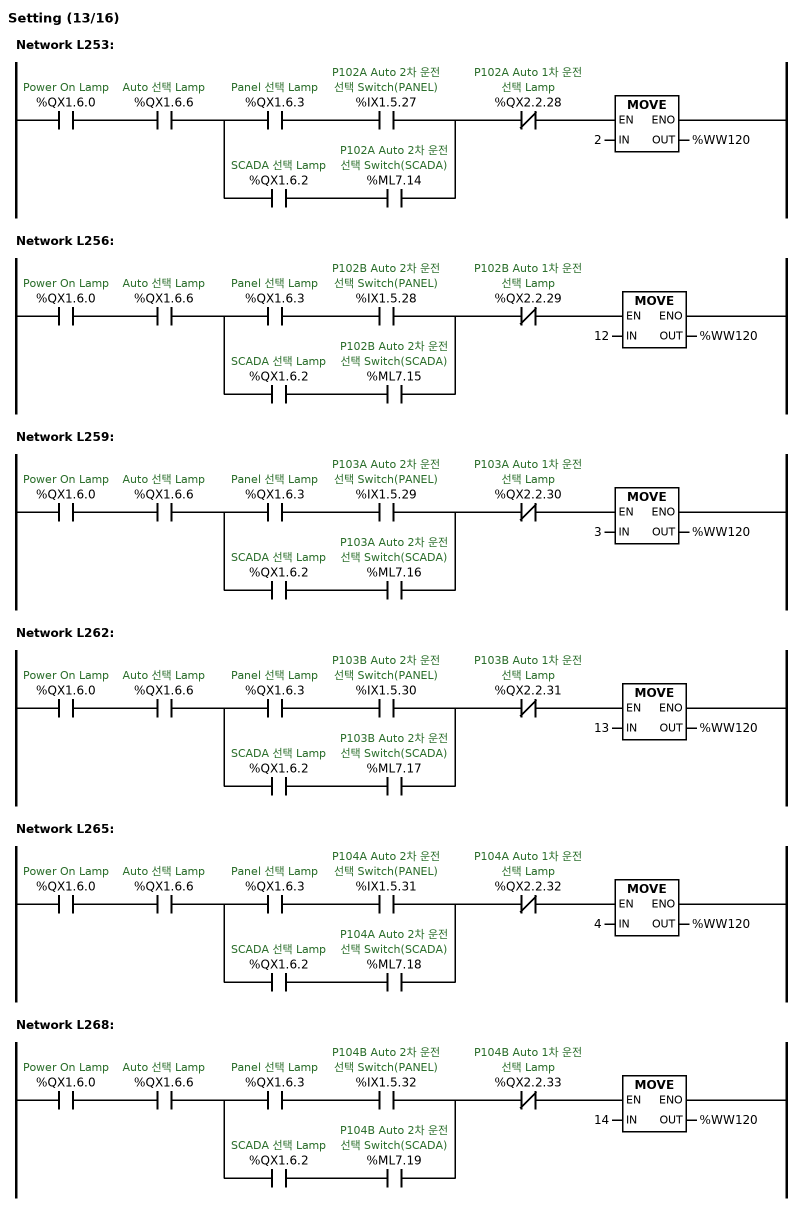
(* [picture p144: Setting rungs L253-L268] *)
(* Rung L253 *)
IF %QX1.6.0 AND %QX1.6.6 AND ((%QX1.6.3 AND %IX1.5.27) OR (%QX1.6.2 AND %ML7.14)) AND NOT %QX2.2.28 THEN
    %WW120 := 2;
END_IF;
(* Rung L256 *)
IF %QX1.6.0 AND %QX1.6.6 AND ((%QX1.6.3 AND %IX1.5.28) OR (%QX1.6.2 AND %ML7.15)) AND NOT %QX2.2.29 THEN
    %WW120 := 12;
END_IF;
(* Rung L259 *)
IF %QX1.6.0 AND %QX1.6.6 AND ((%QX1.6.3 AND %IX1.5.29) OR (%QX1.6.2 AND %ML7.16)) AND NOT %QX2.2.30 THEN
    %WW120 := 3;
END_IF;
(* Rung L262 *)
IF %QX1.6.0 AND %QX1.6.6 AND ((%QX1.6.3 AND %IX1.5.30) OR (%QX1.6.2 AND %ML7.17)) AND NOT %QX2.2.31 THEN
    %WW120 := 13;
END_IF;
(* Rung L265 *)
IF %QX1.6.0 AND %QX1.6.6 AND ((%QX1.6.3 AND %IX1.5.31) OR (%QX1.6.2 AND %ML7.18)) AND NOT %QX2.2.32 THEN
    %WW120 := 4;
END_IF;
(* Rung L268 *)
IF %QX1.6.0 AND %QX1.6.6 AND ((%QX1.6.3 AND %IX1.5.32) OR (%QX1.6.2 AND %ML7.19)) AND NOT %QX2.2.33 THEN
    %WW120 := 14;
END_IF;

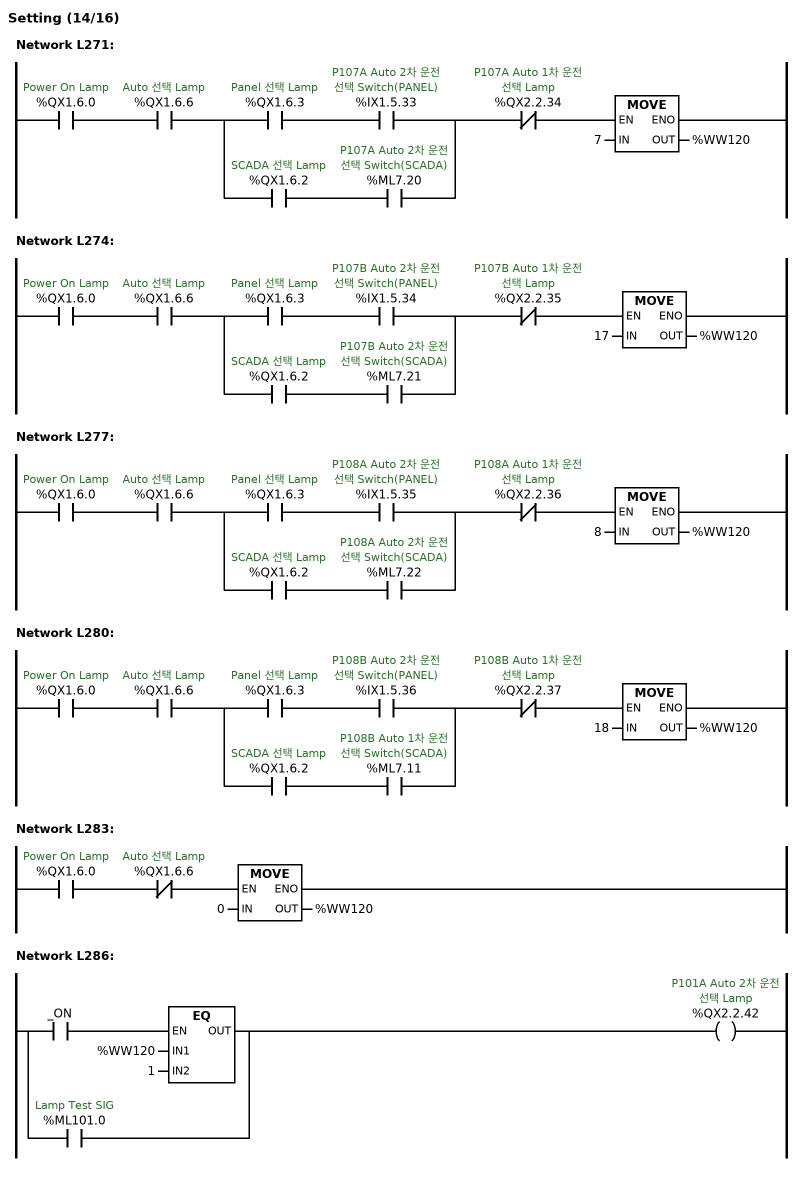
(* Rung L271 *)
IF %QX1.6.0 AND %QX1.6.6 AND ((%QX1.6.3 AND %IX1.5.33) OR (%QX1.6.2 AND %ML7.20)) AND NOT %QX2.2.34 THEN
    %WW120 := 7;
END_IF;
(* Rung L274 *)
IF %QX1.6.0 AND %QX1.6.6 AND ((%QX1.6.3 AND %IX1.5.34) OR (%QX1.6.2 AND %ML7.21)) AND NOT %QX2.2.35 THEN
    %WW120 := 17;
END_IF;
(* Rung L277 *)
IF %QX1.6.0 AND %QX1.6.6 AND ((%QX1.6.3 AND %IX1.5.35) OR (%QX1.6.2 AND %ML7.22)) AND NOT %QX2.2.36 THEN
    %WW120 := 8;
END_IF;
(* Rung L280 *)
IF %QX1.6.0 AND %QX1.6.6 AND ((%QX1.6.3 AND %IX1.5.36) OR (%QX1.6.2 AND %ML7.11)) AND NOT %QX2.2.37 THEN
    %WW120 := 18;
END_IF;
(* Rung L283 *)
IF %QX1.6.0 AND NOT %QX1.6.6 THEN %WW120 := 0; END_IF;
(* Rung L286 *)
IF _ON THEN _t23 := %WW120 = 1; END_IF;
%QX2.2.42 := _t23 OR %ML101.0;

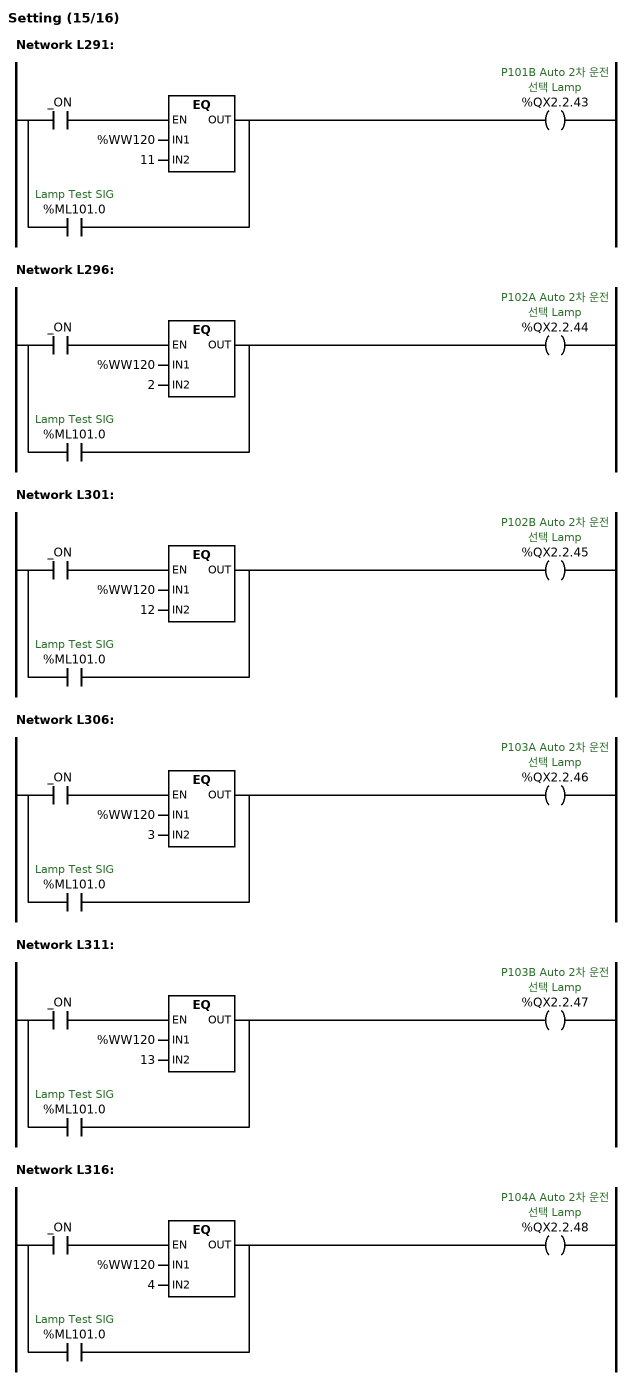
(* Rung L291 *)
IF _ON THEN _t24 := %WW120 = 11; END_IF;
%QX2.2.43 := _t24 OR %ML101.0;
(* Rung L296 *)
IF _ON THEN _t25 := %WW120 = 2; END_IF;
%QX2.2.44 := _t25 OR %ML101.0;
(* Rung L301 *)
IF _ON THEN _t26 := %WW120 = 12; END_IF;
%QX2.2.45 := _t26 OR %ML101.0;
(* Rung L306 *)
IF _ON THEN _t27 := %WW120 = 3; END_IF;
%QX2.2.46 := _t27 OR %ML101.0;
(* Rung L311 *)
IF _ON THEN _t28 := %WW120 = 13; END_IF;
%QX2.2.47 := _t28 OR %ML101.0;
(* Rung L316 *)
IF _ON THEN _t29 := %WW120 = 4; END_IF;
%QX2.2.48 := _t29 OR %ML101.0;

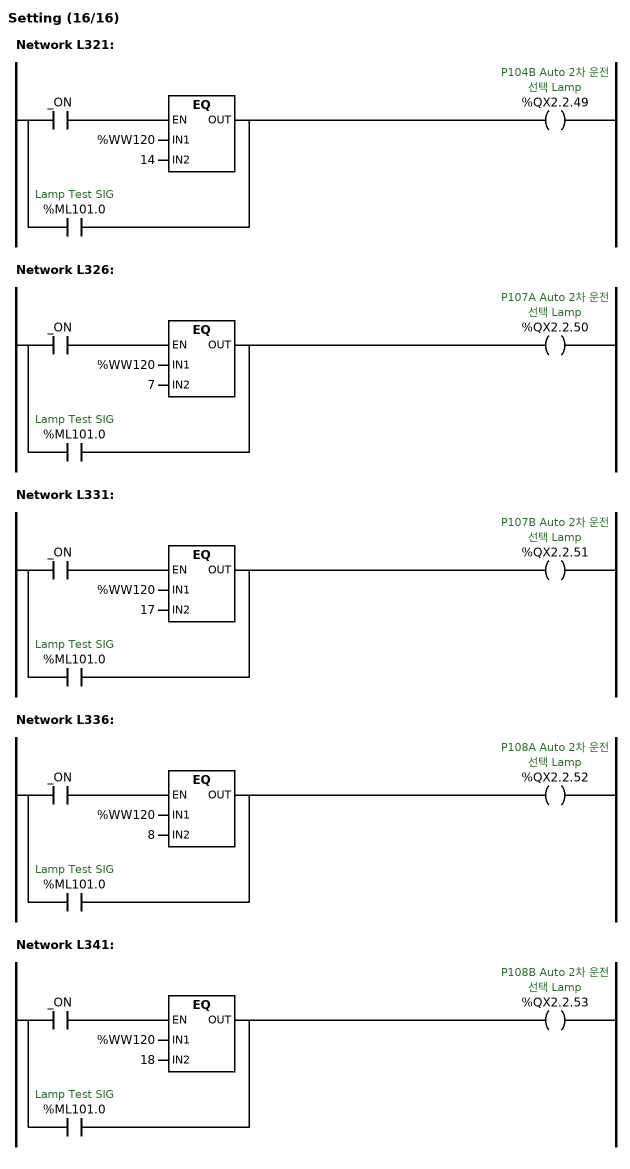
(* Rung L321 *)
IF _ON THEN _t30 := %WW120 = 14; END_IF;
%QX2.2.49 := _t30 OR %ML101.0;
(* Rung L326 *)
IF _ON THEN _t31 := %WW120 = 7; END_IF;
%QX2.2.50 := _t31 OR %ML101.0;
(* Rung L331 *)
IF _ON THEN _t32 := %WW120 = 17; END_IF;
%QX2.2.51 := _t32 OR %ML101.0;
(* Rung L336 *)
IF _ON THEN _t33 := %WW120 = 8; END_IF;
%QX2.2.52 := _t33 OR %ML101.0;
(* Rung L341 *)
IF _ON THEN _t34 := %WW120 = 18; END_IF;
%QX2.2.53 := _t34 OR %ML101.0;
END_PROGRAM

PROGRAM Alarm (* task: 스캔 프로그램 *)
VAR
    _e1 : R_TRIG;
    _e2 : R_TRIG;
    _e3 : R_TRIG;
    _e4 : R_TRIG;
    _e5 : R_TRIG;
    _e6 : R_TRIG;
    _e7 : R_TRIG;
    _e8 : R_TRIG;
END_VAR

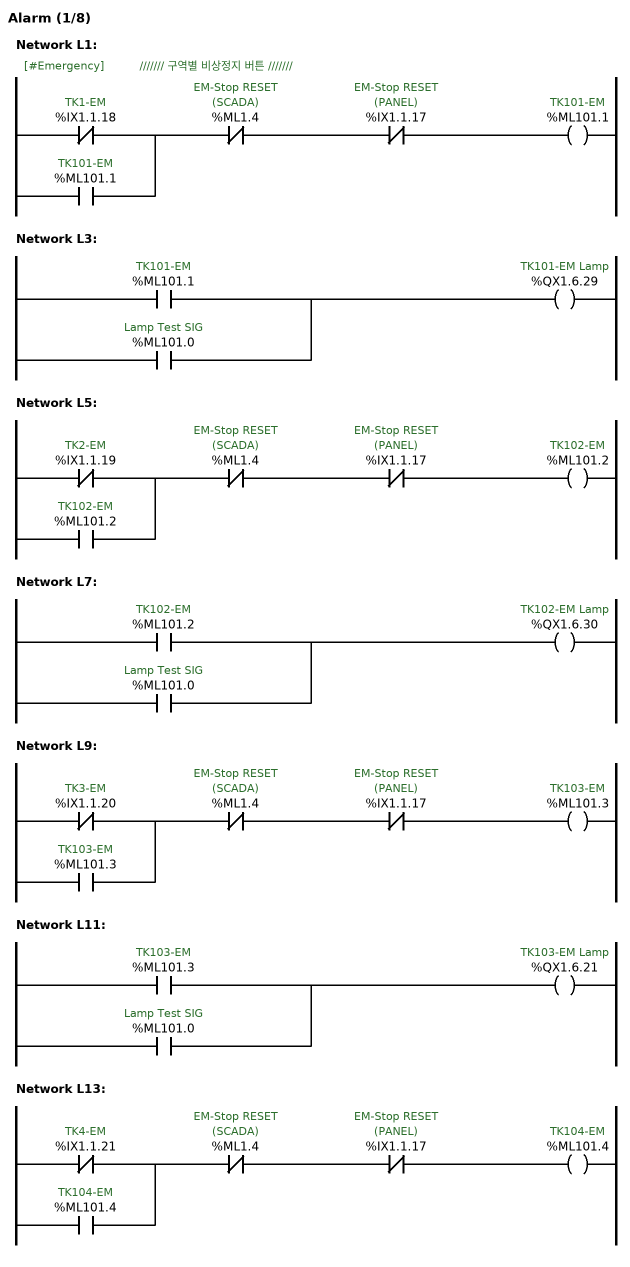
(* [#Emergency]          /////// 구역별 비상정지 버튼 /////// *)
(* Rung L1 *)
%ML101.1 := (NOT %IX1.1.18 OR %ML101.1) AND NOT %ML1.4 AND NOT %IX1.1.17;
(* Rung L3 *)
%QX1.6.29 := %ML101.1 OR %ML101.0;
(* Rung L5 *)
%ML101.2 := (NOT %IX1.1.19 OR %ML101.2) AND NOT %ML1.4 AND NOT %IX1.1.17;
(* Rung L7 *)
%QX1.6.30 := %ML101.2 OR %ML101.0;
(* Rung L9 *)
%ML101.3 := (NOT %IX1.1.20 OR %ML101.3) AND NOT %ML1.4 AND NOT %IX1.1.17;
(* Rung L11 *)
%QX1.6.21 := %ML101.3 OR %ML101.0;
(* Rung L13 *)
%ML101.4 := (NOT %IX1.1.21 OR %ML101.4) AND NOT %ML1.4 AND NOT %IX1.1.17;

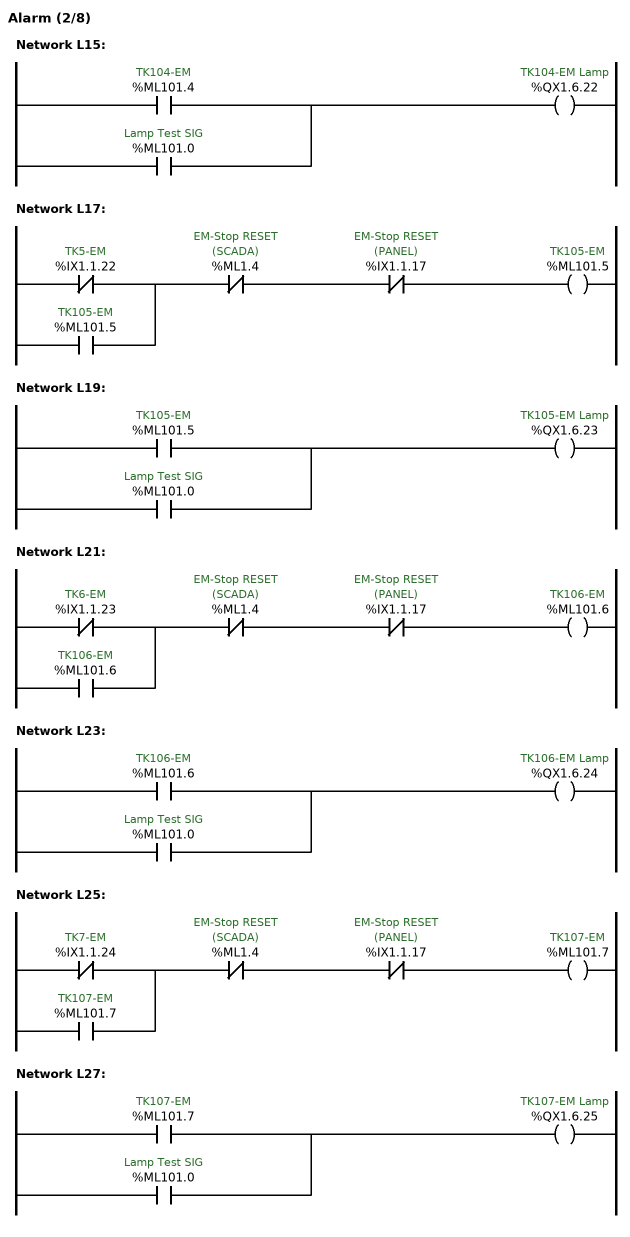
(* Rung L15 *)
%QX1.6.22 := %ML101.4 OR %ML101.0;
(* Rung L17 *)
%ML101.5 := (NOT %IX1.1.22 OR %ML101.5) AND NOT %ML1.4 AND NOT %IX1.1.17;
(* Rung L19 *)
%QX1.6.23 := %ML101.5 OR %ML101.0;
(* Rung L21 *)
%ML101.6 := (NOT %IX1.1.23 OR %ML101.6) AND NOT %ML1.4 AND NOT %IX1.1.17;
(* Rung L23 *)
%QX1.6.24 := %ML101.6 OR %ML101.0;
(* Rung L25 *)
%ML101.7 := (NOT %IX1.1.24 OR %ML101.7) AND NOT %ML1.4 AND NOT %IX1.1.17;
(* Rung L27 *)
%QX1.6.25 := %ML101.7 OR %ML101.0;

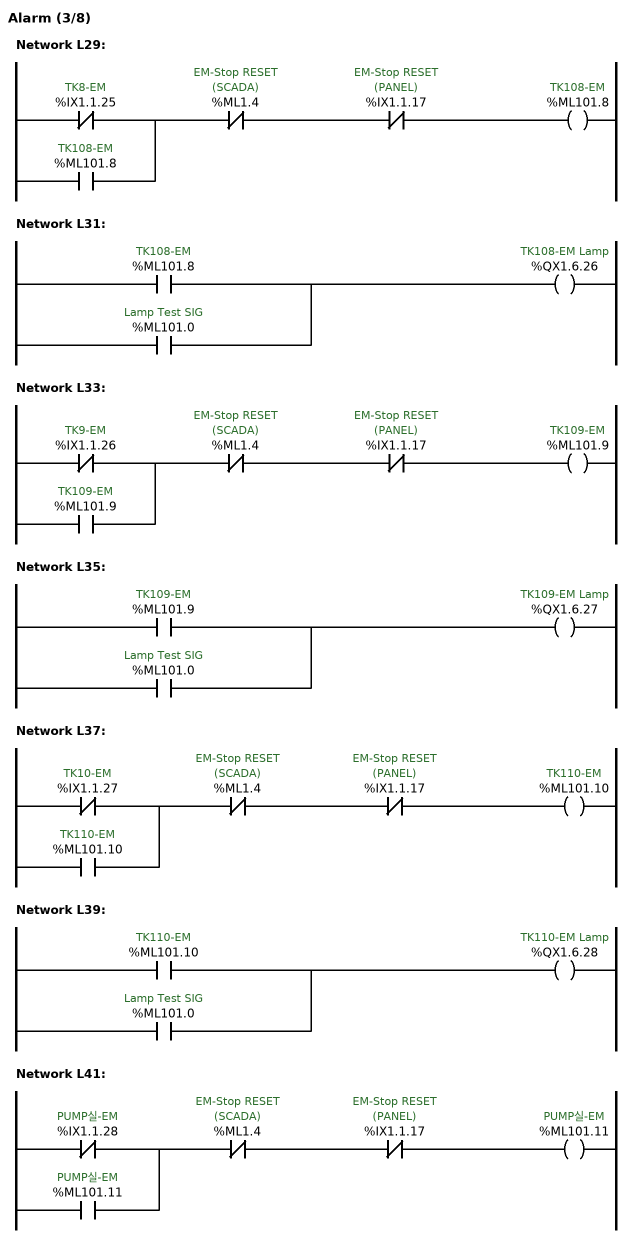
(* Rung L29 *)
%ML101.8 := (NOT %IX1.1.25 OR %ML101.8) AND NOT %ML1.4 AND NOT %IX1.1.17;
(* Rung L31 *)
%QX1.6.26 := %ML101.8 OR %ML101.0;
(* Rung L33 *)
%ML101.9 := (NOT %IX1.1.26 OR %ML101.9) AND NOT %ML1.4 AND NOT %IX1.1.17;
(* Rung L35 *)
%QX1.6.27 := %ML101.9 OR %ML101.0;
(* Rung L37 *)
%ML101.10 := (NOT %IX1.1.27 OR %ML101.10) AND NOT %ML1.4 AND NOT %IX1.1.17;
(* Rung L39 *)
%QX1.6.28 := %ML101.10 OR %ML101.0;
(* Rung L41 *)
%ML101.11 := (NOT %IX1.1.28 OR %ML101.11) AND NOT %ML1.4 AND NOT %IX1.1.17;

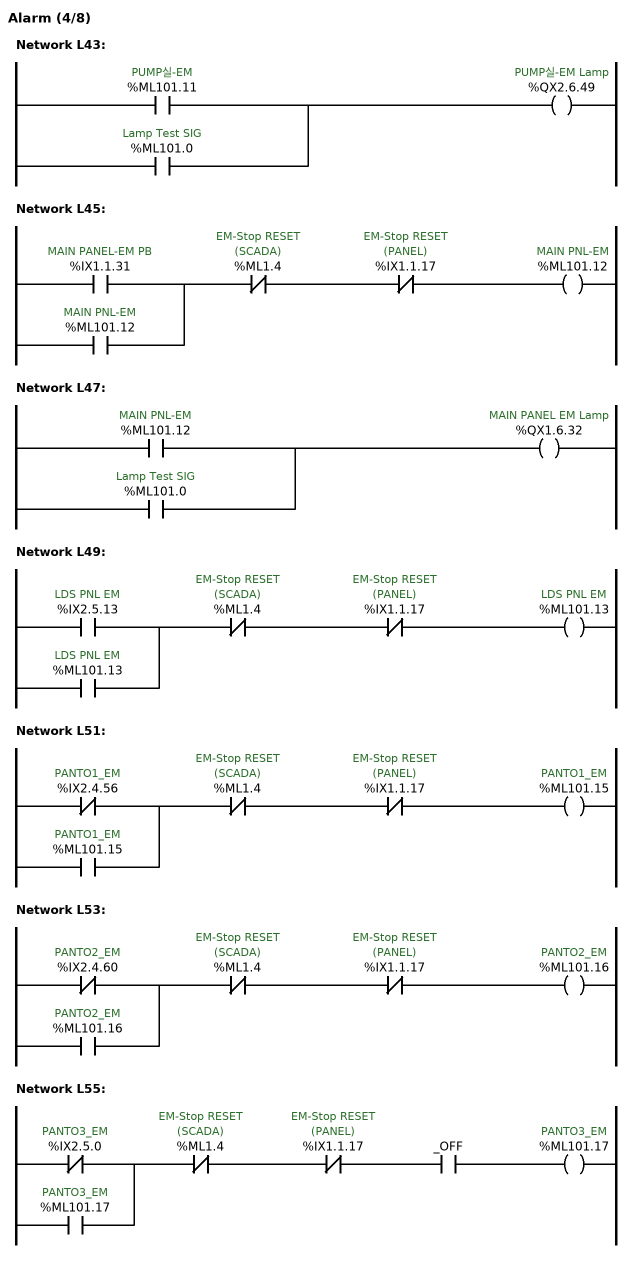
(* Rung L43 *)
%QX2.6.49 := %ML101.11 OR %ML101.0;
(* Rung L45 *)
%ML101.12 := (%IX1.1.31 OR %ML101.12) AND NOT %ML1.4 AND NOT %IX1.1.17;
(* Rung L47 *)
%QX1.6.32 := %ML101.12 OR %ML101.0;
(* Rung L49 *)
%ML101.13 := (%IX2.5.13 OR %ML101.13) AND NOT %ML1.4 AND NOT %IX1.1.17;
(* Rung L51 *)
%ML101.15 := (NOT %IX2.4.56 OR %ML101.15) AND NOT %ML1.4 AND NOT %IX1.1.17;
(* Rung L53 *)
%ML101.16 := (NOT %IX2.4.60 OR %ML101.16) AND NOT %ML1.4 AND NOT %IX1.1.17;
(* Rung L55 *)
%ML101.17 := (NOT %IX2.5.0 OR %ML101.17) AND NOT %ML1.4 AND NOT %IX1.1.17 AND _OFF;

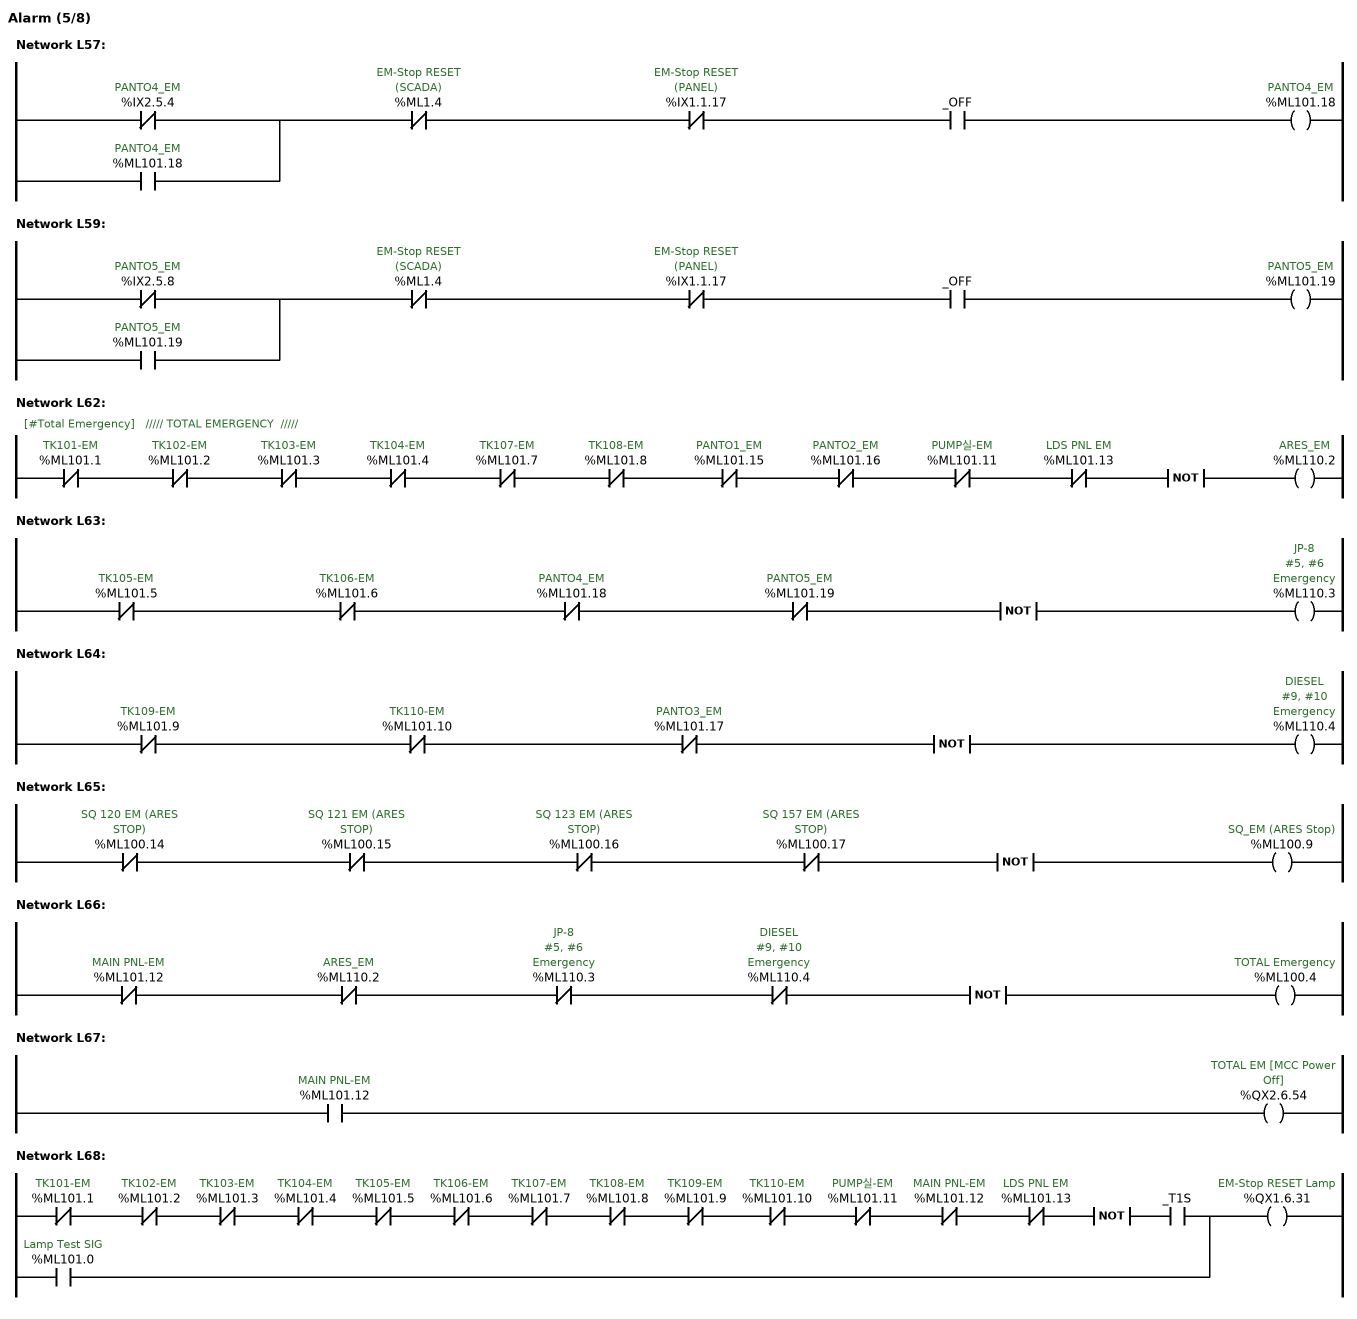
(* Rung L57 *)
%ML101.18 := (NOT %IX2.5.4 OR %ML101.18) AND NOT %ML1.4 AND NOT %IX1.1.17 AND _OFF;
(* Rung L59 *)
%ML101.19 := (NOT %IX2.5.8 OR %ML101.19) AND NOT %ML1.4 AND NOT %IX1.1.17 AND _OFF;
(* [#Total Emergency]   ///// TOTAL EMERGENCY  ///// *)
(* Rung L62 *)
%ML110.2 := NOT (NOT %ML101.1 AND NOT %ML101.2 AND NOT %ML101.3 AND NOT %ML101.4 AND NOT %ML101.7 AND NOT %ML101.8 AND NOT %ML101.15 AND NOT %ML101.16 AND NOT %ML101.11 AND NOT %ML101.13);
(* Rung L63 *)
%ML110.3 := NOT (NOT %ML101.5 AND NOT %ML101.6 AND NOT %ML101.18 AND NOT %ML101.19);
(* Rung L64 *)
%ML110.4 := NOT (NOT %ML101.9 AND NOT %ML101.10 AND NOT %ML101.17);
(* Rung L65 *)
%ML100.9 := NOT (NOT %ML100.14 AND NOT %ML100.15 AND NOT %ML100.16 AND NOT %ML100.17);
(* Rung L66 *)
%ML100.4 := NOT (NOT %ML101.12 AND NOT %ML110.2 AND NOT %ML110.3 AND NOT %ML110.4);
(* Rung L67 *)
%QX2.6.54 := %ML101.12;
(* Rung L68 *)
%QX1.6.31 := (NOT (NOT %ML101.1 AND NOT %ML101.2 AND NOT %ML101.3 AND NOT %ML101.4 AND NOT %ML101.5 AND NOT %ML101.6 AND NOT %ML101.7 AND NOT %ML101.8 AND NOT %ML101.9 AND NOT %ML101.10 AND NOT %ML101.11 AND NOT %ML101.12 AND NOT %ML101.13) AND _T1S) OR %ML101.0;

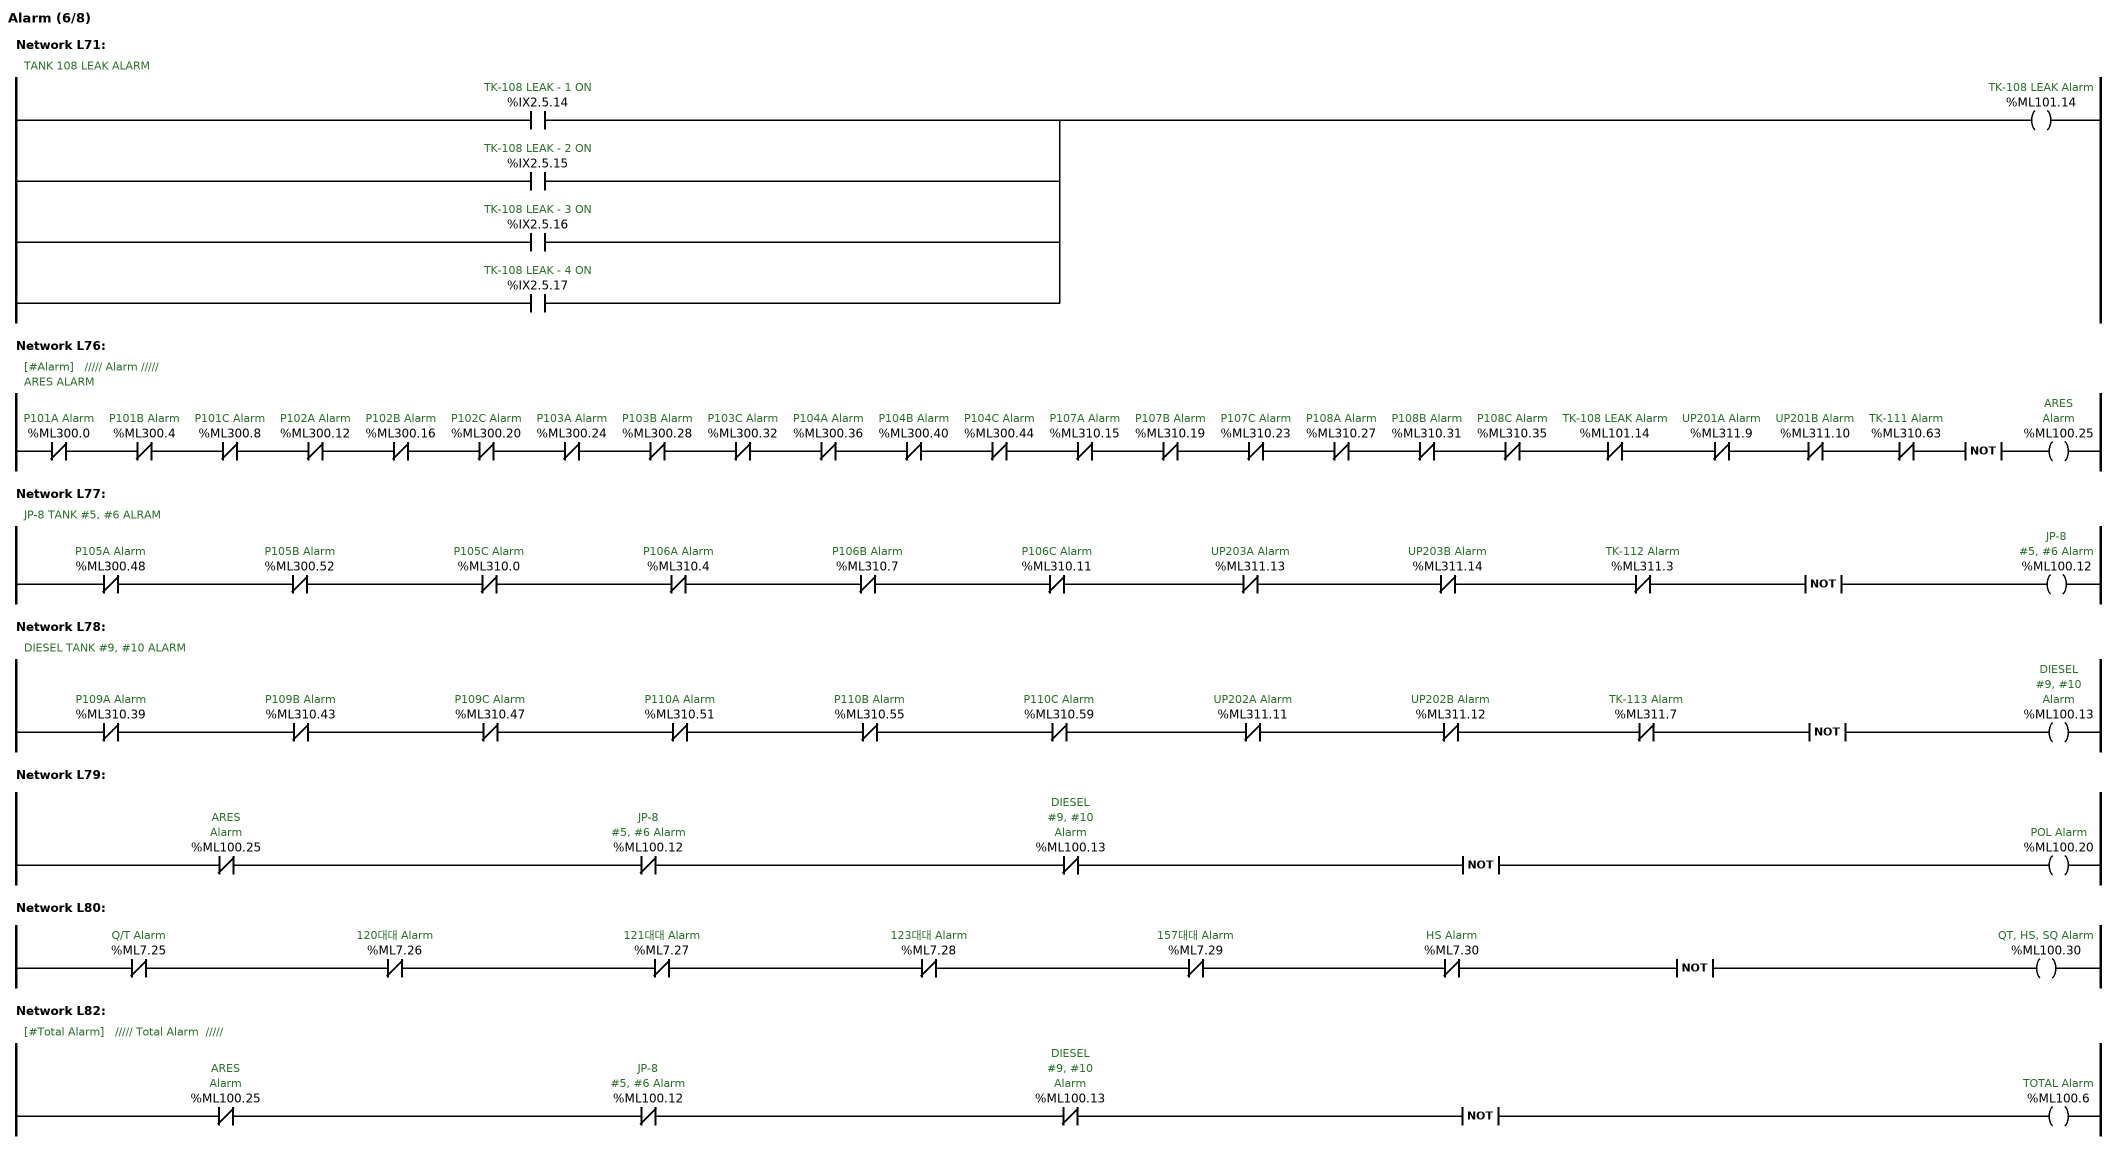
(* TANK 108 LEAK ALARM *)
(* Rung L71 *)
%ML101.14 := %IX2.5.14 OR %IX2.5.15 OR %IX2.5.16 OR %IX2.5.17;
(* [#Alarm]   ///// Alarm ///// *)
(* Rung L76 *)
%ML100.25 := NOT (NOT %ML300.0 AND NOT %ML300.4 AND NOT %ML300.8 AND NOT %ML300.12 AND NOT %ML300.16 AND NOT %ML300.20 AND NOT %ML300.24 AND NOT %ML300.28 AND NOT %ML300.32 AND NOT %ML300.36 AND NOT %ML300.40 AND NOT %ML300.44 AND NOT %ML310.15 AND NOT %ML310.19 AND NOT %ML310.23 AND NOT %ML310.27 AND NOT %ML310.31 AND NOT %ML310.35 AND NOT %ML101.14 AND NOT %ML311.9 AND NOT %ML311.10 AND NOT %ML310.63);
(* ARES ALARM *)
(* Rung L77 *)
%ML100.12 := NOT (NOT %ML300.48 AND NOT %ML300.52 AND NOT %ML310.0 AND NOT %ML310.4 AND NOT %ML310.7 AND NOT %ML310.11 AND NOT %ML311.13 AND NOT %ML311.14 AND NOT %ML311.3);
(* JP-8 TANK #5, #6 ALRAM *)
(* Rung L78 *)
%ML100.13 := NOT (NOT %ML310.39 AND NOT %ML310.43 AND NOT %ML310.47 AND NOT %ML310.51 AND NOT %ML310.55 AND NOT %ML310.59 AND NOT %ML311.11 AND NOT %ML311.12 AND NOT %ML311.7);
(* DIESEL TANK #9, #10 ALARM *)
(* Rung L79 *)
%ML100.20 := NOT (NOT %ML100.25 AND NOT %ML100.12 AND NOT %ML100.13);
(* Rung L80 *)
%ML100.30 := NOT (NOT %ML7.25 AND NOT %ML7.26 AND NOT %ML7.27 AND NOT %ML7.28 AND NOT %ML7.29 AND NOT %ML7.30);
(* [#Total Alarm]   ///// Total Alarm  ///// *)
(* Rung L82 *)
%ML100.6 := NOT (NOT %ML100.25 AND NOT %ML100.12 AND NOT %ML100.13);

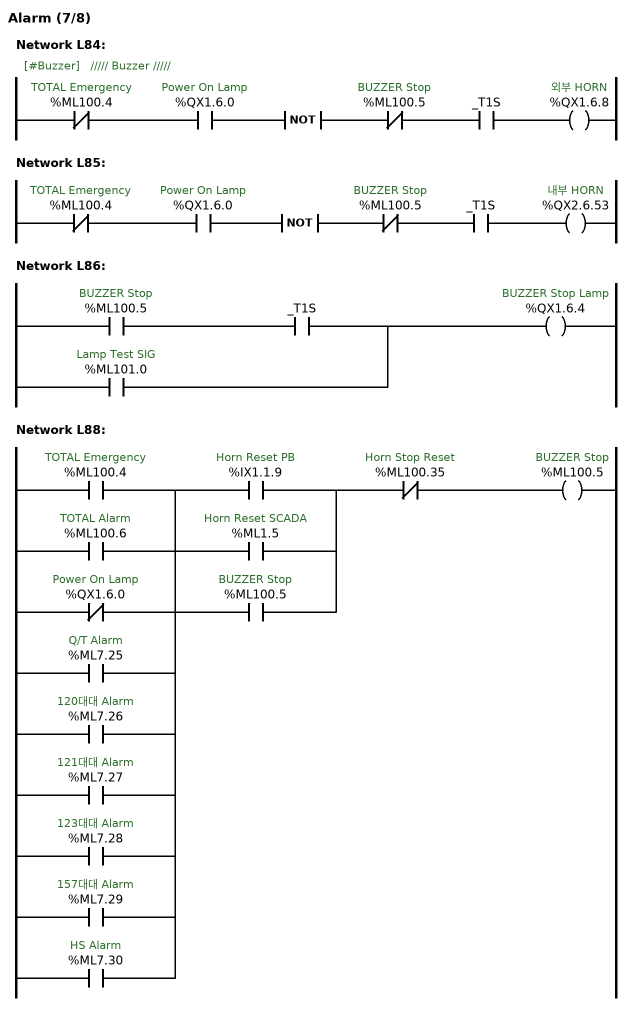
(* [#Buzzer]   ///// Buzzer ///// *)
(* Rung L84 *)
%QX1.6.8 := NOT (NOT %ML100.4 AND %QX1.6.0) AND NOT %ML100.5 AND _T1S;
(* Rung L85 *)
%QX2.6.53 := NOT (NOT %ML100.4 AND %QX1.6.0) AND NOT %ML100.5 AND _T1S;
(* Rung L86 *)
%QX1.6.4 := (%ML100.5 AND _T1S) OR %ML101.0;
(* Rung L88 *)
%ML100.5 := (%ML100.4 OR %ML100.6 OR NOT %QX1.6.0 OR %ML7.25 OR %ML7.26 OR %ML7.27 OR %ML7.28 OR %ML7.29 OR %ML7.30) AND (%IX1.1.9 OR %ML1.5 OR %ML100.5) AND NOT %ML100.35;

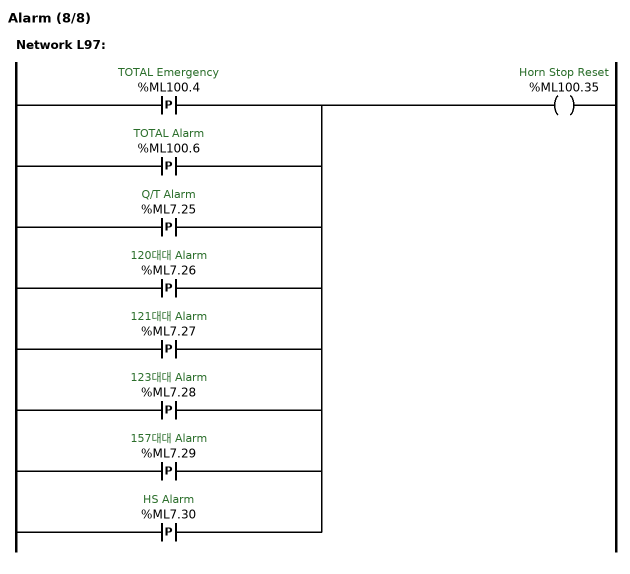
(* Rung L97 *)
_e1(CLK := %ML100.4);
_e2(CLK := %ML100.6);
_e3(CLK := %ML7.25);
_e4(CLK := %ML7.26);
_e5(CLK := %ML7.27);
_e6(CLK := %ML7.28);
_e7(CLK := %ML7.29);
_e8(CLK := %ML7.30);
%ML100.35 := _e1.Q OR _e2.Q OR _e3.Q OR _e4.Q OR _e5.Q OR _e6.Q OR _e7.Q OR _e8.Q;
END_PROGRAM